{attribute 'hide'}
FUNCTION_BLOCK KIN_STATE_OBSERVER_OID_PARAM
VAR_INPUT
	oid														:	UDINT := 0; (* Scara State Observer OID *)
	TooltrafoOID											:	UDINT := 0; (* ToolTrafoOID *)
	NextTrafoOID											:	UDINT := 0; (*StaticTrafoOID *)

END_VAR
VAR_OUTPUT

END_VAR
VAR
END_VAR

;

METHOD delete : BOOL
VAR_INPUT
END_VAR
	oid														:= 0;
	TooltrafoOID											:= 0;
	NextTrafoOID											:= 0;
delete	:= TRUE;
END_METHOD

END_FUNCTION_BLOCK

(* stored: Version 1.1.0.1, ProductVersion 3.1.4024.6
   POU KIN_STATE_OBSERVER_OID_PARAM: Id {d79ddc5d-5ca6-426b-8f4d-a85af5a37d2a}, SpecialFunc None
   Method delete: Id {c5b1b096-648a-487a-aa00-cfba1def4944} *)
